LIN {X 0,Y 119.858,Z 319.555,A -85,B 0,C 180,E1 -30049.333,E2 -30049.333} C_VEL
LIN {X 0,Y 123.743,Z 306.108,A -85,B 0,C 180,E1 -30049.858,E2 -30049.858} C_VEL
LIN {X 0,Y 124.732,Z 301.362,A -85,B 0,C 180,E1 -30050.064,E2 -30050.064} C_VEL
LIN {X 0,Y 124.129,Z 298.09,A -85,B 0,C 180,E1 -30054.11,E2 -30054.11} C_VEL
LIN {X 0,Y 123.862,Z 295.451,A -85,B 0,C 180,E1 -30060,E2 -30060} C_VEL
LIN {X 0,Y 124.197,Z 298.699,A -85,B 0,C 180,E1 -30066.907,E2 -30066.907} C_VEL
LIN {X 0,Y 124.718,Z 301.371,A -85,B 0,C 180,E1 -30070.151,E2 -30070.151} C_VEL
LIN {X 0,Y 121.542,Z 314.132,A -85,B 0,C 180,E1 -30070.596,E2 -30070.596} C_VEL
LIN {X 0,Y 117.209,Z 326.252,A -85,B 0,C 180,E1 -30071.353,E2 -30071.353} C_VEL
LIN {X 0,Y 111.468,Z 338.251,A -85,B 0,C 180,E1 -30072.254,E2 -30072.254} C_VEL
LIN {X 0,Y 104.801,Z 349.276,A -85,B 0,C 180,E1 -30073.511,E2 -30073.511} C_VEL
LIN {X 0,Y 98.169,Z 358.213,A -85,B 0,C 180,E1 -30074.89,E2 -30074.89} C_VEL
LIN {X 0,Y 96.602,Z 360.066,A -85,B 0,C 180,E1 -30075.232,E2 -30075.232} C_VEL
LIN {X 0,Y 92.627,Z 364.399,A -85,B 0,C 180,E1 -30075.737,E2 -30075.737} C_VEL
LIN {X 0,Y 85.256,Z 371.05,A -85,B 0,C 180,E1 -30075.683,E2 -30075.683} C_VEL
LIN {X 0,Y 77.46,Z 377.142,A -85,B 0,C 180,E1 -30075.805,E2 -30075.805} C_VEL
LIN {X 0,Y 72.841,Z 380.518,A -85,B 0,C 180,E1 -30076.777,E2 -30076.777} C_VEL
LIN {X 0,Y 63.694,Z 386.573,A -85,B 0,C 180,E1 -30080.311,E2 -30080.311} C_VEL
LIN {X 0,Y 54.383,Z 391.666,A -85,B 0,C 180,E1 -30085.238,E2 -30085.238} C_VEL
LIN {X 0,Y 45.566,Z 395.622,A -85,B 0,C 180,E1 -30091.98,E2 -30091.98} C_VEL
LIN {X 0,Y 37.753,Z 398.542,A -85,B 0,C 180,E1 -30101.882,E2 -30101.882} C_VEL
LIN {X 0,Y 33.345,Z 399.934,A -85,B 0,C 180,E1 -30110.787,E2 -30110.787} C_VEL
LIN {X 0,Y 29.898,Z 400.925,A -85,B 0,C 180,E1 -30121.964,E2 -30121.964} C_VEL
LIN {X 0,Y 27.084,Z 401.756,A -85,B 0,C 180,E1 -30150.006,E2 -30150.006} C_VEL
LIN {X 0,Y 27.692,Z 401.557,A -85,B 0,C 180,E1 -30164.708,E2 -30164.708} C_VEL
LIN {X 0,Y 29.899,Z 400.965,A -85,B 0,C 180,E1 -30178.048,E2 -30178.048} C_VEL
LIN {X 0,Y 37.747,Z 398.621,A -85,B 0,C 180,E1 -30198.143,E2 -30198.143} C_VEL
LIN {X 0,Y 45.549,Z 395.733,A -85,B 0,C 180,E1 -30208.067,E2 -30208.067} C_VEL
LIN {X 0,Y 54.363,Z 391.816,A -85,B 0,C 180,E1 -30214.822,E2 -30214.822} C_VEL
LIN {X 0,Y 63.677,Z 386.766,A -85,B 0,C 180,E1 -30219.745,E2 -30219.745} C_VEL
LIN {X 0,Y 73.296,Z 380.406,A -85,B 0,C 180,E1 -30223.511,E2 -30223.511} C_VEL
LIN {X 0,Y 83.126,Z 372.457,A -85,B 0,C 180,E1 -30226.482,E2 -30226.482} C_VEL
LIN {X 0,Y 93.192,Z 362.567,A -85,B 0,C 180,E1 -30228.636,E2 -30228.636} C_VEL
LIN {X 0,Y 101.655,Z 352.177,A -85,B 0,C 180,E1 -30230.129,E2 -30230.129} C_VEL
LIN {X 0,Y 109.313,Z 340.466,A -85,B 0,C 180,E1 -30231.304,E2 -30231.304} C_VEL
LIN {X 0,Y 115.288,Z 328.776,A -85,B 0,C 180,E1 -30232.11,E2 -30232.11} C_VEL
LIN {X 0,Y 119.884,Z 316.966,A -85,B 0,C 180,E1 -30232.67,E2 -30232.67} C_VEL
LIN {X 0,Y 122.909,Z 306.336,A -85,B 0,C 180,E1 -30233.121,E2 -30233.121} C_VEL
LIN {X 0,Y 122.769,Z 304.591,A -85,B 0,C 180,E1 -30235.896,E2 -30235.896} C_VEL
LIN {X 0,Y 122.833,Z 303.055,A -85,B 0,C 180,E1 -30240,E2 -30240} C_VEL
LIN {X 0,Y 122.855,Z 305.465,A -85,B 0,C 180,E1 -30245.539,E2 -30245.539} C_VEL
LIN {X 0,Y 122.934,Z 306.392,A -85,B 0,C 180,E1 -30246.818,E2 -30246.818} C_VEL
LIN {X 0,Y 119.051,Z 319.603,A -85,B 0,C 180,E1 -30247.302,E2 -30247.302} C_VEL
LIN {X 0,Y 114.106,Z 331.478,A -85,B 0,C 180,E1 -30247.858,E2 -30247.858} C_VEL
LIN {X 0,Y 107.541,Z 343.596,A -85,B 0,C 180,E1 -30248.716,E2 -30248.716} C_VEL
LIN {X 0,Y 99.871,Z 354.762,A -85,B 0,C 180,E1 -30249.87,E2 -30249.87} C_VEL
LIN {X 0,Y 91.405,Z 364.671,A -85,B 0,C 180,E1 -30251.38,E2 -30251.38} C_VEL
LIN {X 0,Y 81.351,Z 374.276,A -85,B 0,C 180,E1 -30253.61,E2 -30253.61} C_VEL
LIN {X 0,Y 71.482,Z 381.916,A -85,B 0,C 180,E1 -30256.539,E2 -30256.539} C_VEL
LIN {X 0,Y 62.526,Z 387.71,A -85,B 0,C 180,E1 -30260.241,E2 -30260.241} C_VEL
LIN {X 0,Y 51.135,Z 393.654,A -85,B 0,C 180,E1 -30266.698,E2 -30266.698} C_VEL
LIN {X 0,Y 42.552,Z 397.231,A -85,B 0,C 180,E1 -30274.324,E2 -30274.324} C_VEL
LIN {X 0,Y 37.428,Z 399.073,A -85,B 0,C 180,E1 -30281.309,E2 -30281.309} C_VEL
LIN {X 0,Y 29.679,Z 401.443,A -85,B 0,C 180,E1 -30301.726,E2 -30301.726} C_VEL
LIN {X 0,Y 27.578,Z 402.044,A -85,B 0,C 180,E1 -30315.23,E2 -30315.23} C_VEL
LIN {X 0,Y 27.017,Z 402.251,A -85,B 0,C 180,E1 -30329.994,E2 -30329.994} C_VEL
LIN {X 0,Y 27.577,Z 402.023,A -85,B 0,C 180,E1 -30344.758,E2 -30344.758} C_VEL
LIN {X 0,Y 29.678,Z 401.408,A -85,B 0,C 180,E1 -30358.262,E2 -30358.262} C_VEL
LIN {X 0,Y 33.057,Z 400.407,A -85,B 0,C 180,E1 -30369.62,E2 -30369.62} C_VEL
LIN {X 0,Y 37.427,Z 399.003,A -85,B 0,C 180,E1 -30378.679,E2 -30378.679} C_VEL
LIN {X 0,Y 45.329,Z 396.066,A -85,B 0,C 180,E1 -30388.501,E2 -30388.501} C_VEL
LIN {X 0,Y 54.111,Z 392.092,A -85,B 0,C 180,E1 -30395.381,E2 -30395.381} C_VEL
LIN {X 0,Y 64.611,Z 386.273,A -85,B 0,C 180,E1 -30400.708,E2 -30400.708} C_VEL
LIN {X 0,Y 74.738,Z 379.307,A -85,B 0,C 180,E1 -30404.536,E2 -30404.536} C_VEL
LIN {X 0,Y 84.675,Z 371.03,A -85,B 0,C 180,E1 -30407.209,E2 -30407.209} C_VEL
LIN {X 0,Y 93.082,Z 362.531,A -85,B 0,C 180,E1 -30408.959,E2 -30408.959} C_VEL
LIN {X 0,Y 101.56,Z 352.031,A -85,B 0,C 180,E1 -30410.418,E2 -30410.418} C_VEL
LIN {X 0,Y 109.251,Z 340.203,A -85,B 0,C 180,E1 -30411.496,E2 -30411.496} C_VEL
LIN {X 0,Y 115.146,Z 328.502,A -85,B 0,C 180,E1 -30412.244,E2 -30412.244} C_VEL
LIN {X 0,Y 119.879,Z 316.102,A -85,B 0,C 180,E1 -30412.807,E2 -30412.807} C_VEL
LIN {X 0,Y 122.665,Z 306.102,A -85,B 0,C 180,E1 -30413.163,E2 -30413.163} C_VEL
LIN {X 0,Y 122.509,Z 304.37,A -85,B 0,C 180,E1 -30415.888,E2 -30415.888} C_VEL
LIN {X 0,Y 122.58,Z 302.578,A -85,B 0,C 180,E1 -30420,E2 -30420} C_VEL
LIN {X 0,Y 122.58,Z 305.293,A -85,B 0,C 180,E1 -30425.965,E2 -30425.965} C_VEL
LIN {X 0,Y 122.633,Z 306.102,A -85,B 0,C 180,E1 -30427.013,E2 -30427.013} C_VEL
LIN {X 0,Y 119.005,Z 318.553,A -85,B 0,C 180,E1 -30427.448,E2 -30427.448} C_VEL
LIN {X 0,Y 114.142,Z 330.578,A -85,B 0,C 180,E1 -30428.163,E2 -30428.163} C_VEL
LIN {X 0,Y 108.476,Z 341.312,A -85,B 0,C 180,E1 -30428.895,E2 -30428.895} C_VEL
LIN {X 0,Y 100.82,Z 352.87,A -85,B 0,C 180,E1 -30430.075,E2 -30430.075} C_VEL
LIN {X 0,Y 93.211,Z 362.184,A -85,B 0,C 180,E1 -30431.441,E2 -30431.441} C_VEL
LIN {X 0,Y 84.828,Z 370.668,A -85,B 0,C 180,E1 -30433.238,E2 -30433.238} C_VEL
LIN {X 0,Y 74.96,Z 378.924,A -85,B 0,C 180,E1 -30436.065,E2 -30436.065} C_VEL
LIN {X 0,Y 72.841,Z 380.518,A -85,B 0,C 180,E1 -30436.777,E2 -30436.777} C_VEL
LIN {X 0,Y 68.081,Z 383.726,A -85,B 0,C 180,E1 -30437.92,E2 -30437.92} C_VEL
LIN {X 0,Y 59.396,Z 388.459,A -85,B 0,C 180,E1 -30438.633,E2 -30438.633} C_VEL
LIN {X 0,Y 50.354,Z 392.477,A -85,B 0,C 180,E1 -30439.651,E2 -30439.651} C_VEL
LIN {X 0,Y 45.103,Z 394.564,A -85,B 0,C 180,E1 -30441.793,E2 -30441.793} C_VEL
LIN {X 0,Y 39.18,Z 396.752,A -85,B 0,C 180,E1 -30446.263,E2 -30446.263} C_VEL
LIN {X 0,Y 33.422,Z 398.607,A -85,B 0,C 180,E1 -30452.752,E2 -30452.752} C_VEL
LIN {X 0,Y 28.201,Z 400,A -85,B 0,C 180,E1 -30461.625,E2 -30461.625} C_VEL
LIN {X 0,Y 23.871,Z 400.99,A -85,B 0,C 180,E1 -30473.936,E2 -30473.936} C_VEL
LIN {X 0,Y 19.993,Z 401.821,A -85,B 0,C 180,E1 -30510.009,E2 -30510.009} C_VEL
LIN {X 0,Y 20.915,Z 401.621,A -85,B 0,C 180,E1 -30529.643,E2 -30529.643} C_VEL
LIN {X 0,Y 23.872,Z 401.029,A -85,B 0,C 180,E1 -30546.08,E2 -30546.08} C_VEL
LIN {X 0,Y 33.417,Z 398.686,A -85,B 0,C 180,E1 -30567.279,E2 -30567.279} C_VEL
LIN {X 0,Y 42.218,Z 395.798,A -85,B 0,C 180,E1 -30576.294,E2 -30576.294} C_VEL
LIN {X 0,Y 51.737,Z 391.88,A -85,B 0,C 180,E1 -30581.974,E2 -30581.974} C_VEL
LIN {X 0,Y 61.581,Z 386.83,A -85,B 0,C 180,E1 -30585.953,E2 -30585.953} C_VEL
LIN {X 0,Y 71.602,Z 380.47,A -85,B 0,C 180,E1 -30588.98,E2 -30588.98} C_VEL
LIN {X 0,Y 81.756,Z 372.52,A -85,B 0,C 180,E1 -30591.338,E2 -30591.338} C_VEL
LIN {X 0,Y 92.055,Z 362.629,A -85,B 0,C 180,E1 -30592.982,E2 -30592.982} C_VEL
LIN {X 0,Y 100.681,Z 352.239,A -85,B 0,C 180,E1 -30594.111,E2 -30594.111} C_VEL
LIN {X 0,Y 108.466,Z 340.526,A -85,B 0,C 180,E1 -30595.019,E2 -30595.019} C_VEL
LIN {X 0,Y 114.706,Z 328.435,A -85,B 0,C 180,E1 -30595.637,E2 -30595.637} C_VEL
LIN {X 0,Y 119.751,Z 315.33,A -85,B 0,C 180,E1 -30596.116,E2 -30596.116} C_VEL
LIN {X 0,Y 120.925,Z 311.412,A -85,B 0,C 180,E1 -30596.328,E2 -30596.328} C_VEL
LIN {X 0,Y 121.08,Z 310.072,A -85,B 0,C 180,E1 -30600,E2 -30600} C_VEL
LIN {X 0,Y 120.94,Z 311.447,A -85,B 0,C 180,E1 -30603.605,E2 -30603.605} C_VEL
LIN {X 0,Y 116.62,Z 324.08,A -85,B 0,C 180,E1 -30604.065,E2 -30604.065} C_VEL
LIN {X 0,Y 111.907,Z 334.363,A -85,B 0,C 180,E1 -30604.448,E2 -30604.448} C_VEL
LIN {X 0,Y 104.96,Z 346.241,A -85,B 0,C 180,E1 -30605.113,E2 -30605.113} C_VEL
LIN {X 0,Y 97.171,Z 356.84,A -85,B 0,C 180,E1 -30606.016,E2 -30606.016} C_VEL
LIN {X 0,Y 88.549,Z 366.391,A -85,B 0,C 180,E1 -30607.2,E2 -30607.2} C_VEL
LIN {X 0,Y 78.271,Z 375.58,A -85,B 0,C 180,E1 -30608.991,E2 -30608.991} C_VEL
LIN {X 0,Y 68.112,Z 382.971,A -85,B 0,C 180,E1 -30611.403,E2 -30611.403} C_VEL
LIN {X 0,Y 58.133,Z 388.905,A -85,B 0,C 180,E1 -30614.719,E2 -30614.719} C_VEL
LIN {X 0,Y 48.353,Z 393.59,A -85,B 0,C 180,E1 -30619.127,E2 -30619.127} C_VEL
LIN {X 0,Y 38.99,Z 397.167,A -85,B 0,C 180,E1 -30625.67,E2 -30625.67} C_VEL
LIN {X 0,Y 33.154,Z 399.009,A -85,B 0,C 180,E1 -30632.007,E2 -30632.007} C_VEL
LIN {X 0,Y 23.66,Z 401.378,A -85,B 0,C 180,E1 -30653.545,E2 -30653.545} C_VEL
LIN {X 0,Y 20.788,Z 401.979,A -85,B 0,C 180,E1 -30670.232,E2 -30670.232} C_VEL
LIN {X 0,Y 19.936,Z 402.186,A -85,B 0,C 180,E1 -30689.991,E2 -30689.991} C_VEL
LIN {X 0,Y 20.787,Z 401.957,A -85,B 0,C 180,E1 -30709.752,E2 -30709.752} C_VEL
LIN {X 0,Y 23.658,Z 401.342,A -85,B 0,C 180,E1 -30726.44,E2 -30726.44} C_VEL
LIN {X 0,Y 27.941,Z 400.341,A -85,B 0,C 180,E1 -30738.978,E2 -30738.978} C_VEL
LIN {X 0,Y 33.152,Z 398.937,A -85,B 0,C 180,E1 -30747.981,E2 -30747.981} C_VEL
LIN {X 0,Y 42.044,Z 395.999,A -85,B 0,C 180,E1 -30756.82,E2 -30756.82} C_VEL
LIN {X 0,Y 51.554,Z 392.026,A -85,B 0,C 180,E1 -30762.588,E2 -30762.588} C_VEL
LIN {X 0,Y 61.869,Z 386.661,A -85,B 0,C 180,E1 -30766.619,E2 -30766.619} C_VEL
LIN {X 0,Y 71.468,Z 380.473,A -85,B 0,C 180,E1 -30769.516,E2 -30769.516} C_VEL
LIN {X 0,Y 81.679,Z 372.449,A -85,B 0,C 180,E1 -30771.669,E2 -30771.669} C_VEL
LIN {X 0,Y 90.263,Z 364.268,A -85,B 0,C 180,E1 -30773.063,E2 -30773.063} C_VEL
LIN {X 0,Y 98.887,Z 354.286,A -85,B 0,C 180,E1 -30774.232,E2 -30774.232} C_VEL
LIN {X 0,Y 106.695,Z 342.991,A -85,B 0,C 180,E1 -30775.023,E2 -30775.023} C_VEL
LIN {X 0,Y 112.768,Z 331.918,A -85,B 0,C 180,E1 -30775.644,E2 -30775.644} C_VEL
LIN {X 0,Y 117.87,Z 319.915,A -85,B 0,C 180,E1 -30776.106,E2 -30776.106} C_VEL
LIN {X 0,Y 120.679,Z 311.152,A -85,B 0,C 180,E1 -30776.382,E2 -30776.382} C_VEL
LIN {X 0,Y 120.856,Z 309.624,A -85,B 0,C 180,E1 -30780,E2 -30780} C_VEL
LIN {X 0,Y 120.636,Z 311.232,A -85,B 0,C 180,E1 -30783.818,E2 -30783.818} C_VEL
LIN {X 0,Y 116.339,Z 323.817,A -85,B 0,C 180,E1 -30784.28,E2 -30784.28} C_VEL
LIN {X 0,Y 111.077,Z 335.229,A -85,B 0,C 180,E1 -30784.815,E2 -30784.815} C_VEL
LIN {X 0,Y 104.142,Z 346.85,A -85,B 0,C 180,E1 -30785.527,E2 -30785.527} C_VEL
LIN {X 0,Y 96.37,Z 357.295,A -85,B 0,C 180,E1 -30786.494,E2 -30786.494} C_VEL
LIN {X 0,Y 88.629,Z 365.833,A -85,B 0,C 180,E1 -30787.628,E2 -30787.628} C_VEL
LIN {X 0,Y 80.081,Z 373.701,A -85,B 0,C 180,E1 -30789.159,E2 -30789.159} C_VEL
LIN {X 0,Y 70.057,Z 381.313,A -85,B 0,C 180,E1 -30791.575,E2 -30791.575} C_VEL
LIN {X 0,Y 61.592,Z 386.64,A -85,B 0,C 180,E1 -30794.112,E2 -30794.112} C_VEL
LIN {X 0,Y 51.757,Z 391.732,A -85,B 0,C 180,E1 -30798.114,E2 -30798.114} C_VEL
LIN {X 0,Y 45.103,Z 394.564,A -85,B 0,C 180,E1 -30801.793,E2 -30801.793} C_VEL
LIN {X 0,Y 39.871,Z 396.435,A -85,B 0,C 180,E1 -30804.577,E2 -30804.577} C_VEL
LIN {X 0,Y 30.579,Z 398.907,A -85,B 0,C 180,E1 -30808.552,E2 -30808.552} C_VEL
LIN {X 0,Y 23.152,Z 400.348,A -85,B 0,C 180,E1 -30813.818,E2 -30813.818} C_VEL
LIN {X 0,Y 18.175,Z 401.13,A -85,B 0,C 180,E1 -30822.554,E2 -30822.554} C_VEL
LIN {X 0,Y 16.811,Z 401.283,A -85,B 0,C 180,E1 -30827.195,E2 -30827.195} C_VEL
LIN {X 0,Y 12.914,Z 401.886,A -85,B 0,C 180,E1 -30870.013,E2 -30870.013} C_VEL
LIN {X 0,Y 14.424,Z 401.686,A -85,B 0,C 180,E1 -30899.173,E2 -30899.173} C_VEL
LIN {X 0,Y 18.598,Z 401.094,A -85,B 0,C 180,E1 -30919.108,E2 -30919.108} C_VEL
LIN {X 0,Y 30.17,Z 398.75,A -85,B 0,C 180,E1 -30938.726,E2 -30938.726} C_VEL
LIN {X 0,Y 39.893,Z 395.862,A -85,B 0,C 180,E1 -30945.694,E2 -30945.694} C_VEL
LIN {X 0,Y 49.995,Z 391.944,A -85,B 0,C 180,E1 -30949.753,E2 -30949.753} C_VEL
LIN {X 0,Y 60.252,Z 386.893,A -85,B 0,C 180,E1 -30952.519,E2 -30952.519} C_VEL
LIN {X 0,Y 70.587,Z 380.533,A -85,B 0,C 180,E1 -30954.663,E2 -30954.663} C_VEL
LIN {X 0,Y 80.991,Z 372.582,A -85,B 0,C 180,E1 -30956.309,E2 -30956.309} C_VEL
LIN {X 0,Y 91.459,Z 362.692,A -85,B 0,C 180,E1 -30957.404,E2 -30957.404} C_VEL
LIN {X 0,Y 100.202,Z 352.3,A -85,B 0,C 180,E1 -30958.148,E2 -30958.148} C_VEL
LIN {X 0,Y 108.081,Z 340.587,A -85,B 0,C 180,E1 -30958.771,E2 -30958.771} C_VEL
LIN {X 0,Y 113.837,Z 329.724,A -85,B 0,C 180,E1 -30959.144,E2 -30959.144} C_VEL
LIN {X 0,Y 118.639,Z 317.882,A -85,B 0,C 180,E1 -30959.442,E2 -30959.442} C_VEL
LIN {X 0,Y 118.928,Z 317.019,A -85,B 0,C 180,E1 -30959.577,E2 -30959.577} C_VEL
LIN {X 0,Y 118.908,Z 317.083,A -85,B 0,C 180,E1 -30960.222,E2 -30960.222} C_VEL
LIN {X 0,Y 118.089,Z 319.488,A -85,B 0,C 180,E1 -30960.447,E2 -30960.447} C_VEL
LIN {X 0,Y 113.146,Z 331.152,A -85,B 0,C 180,E1 -30960.689,E2 -30960.689} C_VEL
LIN {X 0,Y 106.32,Z 343.476,A -85,B 0,C 180,E1 -30961.143,E2 -30961.143} C_VEL
LIN {X 0,Y 98.436,Z 354.639,A -85,B 0,C 180,E1 -30961.702,E2 -30961.702} C_VEL
LIN {X 0,Y 89.69,Z 364.546,A -85,B 0,C 180,E1 -30962.456,E2 -30962.456} C_VEL
LIN {X 0,Y 80.962,Z 372.67,A -85,B 0,C 180,E1 -30963.363,E2 -30963.363} C_VEL
LIN {X 0,Y 70.529,Z 380.643,A -85,B 0,C 180,E1 -30964.799,E2 -30964.799} C_VEL
LIN {X 0,Y 59.698,Z 387.279,A -85,B 0,C 180,E1 -30966.991,E2 -30966.991} C_VEL
LIN {X 0,Y 49.897,Z 392.099,A -85,B 0,C 180,E1 -30969.603,E2 -30969.603} C_VEL
LIN {X 0,Y 39.789,Z 396.036,A -85,B 0,C 180,E1 -30973.708,E2 -30973.708} C_VEL
LIN {X 0,Y 29.991,Z 398.944,A -85,B 0,C 180,E1 -30980.374,E2 -30980.374} C_VEL
LIN {X 0,Y 18.419,Z 401.313,A -85,B 0,C 180,E1 -31000.246,E2 -31000.246} C_VEL
LIN {X 0,Y 14.295,Z 401.914,A -85,B 0,C 180,E1 -31020.538,E2 -31020.538} C_VEL
LIN {X 0,Y 12.841,Z 402.121,A -85,B 0,C 180,E1 -31049.986,E2 -31049.986} C_VEL
LIN {X 0,Y 14.292,Z 401.892,A -85,B 0,C 180,E1 -31079.44,E2 -31079.44} C_VEL
LIN {X 0,Y 18.416,Z 401.277,A -85,B 0,C 180,E1 -31099.737,E2 -31099.737} C_VEL
LIN {X 0,Y 23.881,Z 400.275,A -85,B 0,C 180,E1 -31111.973,E2 -31111.973} C_VEL
LIN {X 0,Y 29.986,Z 398.871,A -85,B 0,C 180,E1 -31119.615,E2 -31119.615} C_VEL
LIN {X 0,Y 39.783,Z 395.933,A -85,B 0,C 180,E1 -31126.294,E2 -31126.294} C_VEL
LIN {X 0,Y 49.89,Z 391.96,A -85,B 0,C 180,E1 -31130.403,E2 -31130.403} C_VEL
LIN {X 0,Y 61.488,Z 386.08,A -85,B 0,C 180,E1 -31133.437,E2 -31133.437} C_VEL
LIN {X 0,Y 72.255,Z 379.173,A -85,B 0,C 180,E1 -31135.496,E2 -31135.496} C_VEL
LIN {X 0,Y 82.698,Z 370.895,A -85,B 0,C 180,E1 -31136.867,E2 -31136.867} C_VEL
LIN {X 0,Y 91.43,Z 362.395,A -85,B 0,C 180,E1 -31137.744,E2 -31137.744} C_VEL
LIN {X 0,Y 100.18,Z 351.893,A -85,B 0,C 180,E1 -31138.463,E2 -31138.463} C_VEL
LIN {X 0,Y 108.068,Z 340.063,A -85,B 0,C 180,E1 -31138.958,E2 -31138.958} C_VEL
LIN {X 0,Y 114.469,Z 327.524,A -85,B 0,C 180,E1 -31139.342,E2 -31139.342} C_VEL
LIN {X 0,Y 118.391,Z 317.575,A -85,B 0,C 180,E1 -31139.587,E2 -31139.587} C_VEL
LIN {X 0,Y 118.725,Z 316.57,A -85,B 0,C 180,E1 -31140,E2 -31140} C_VEL
LIN {X 0,Y 118.692,Z 316.668,A -85,B 0,C 180,E1 -31140.424,E2 -31140.424} C_VEL
LIN {X 0,Y 116.544,Z 322.553,A -85,B 0,C 180,E1 -31140.733,E2 -31140.733} C_VEL
LIN {X 0,Y 111.585,Z 333.578,A -85,B 0,C 180,E1 -31141.111,E2 -31141.111} C_VEL
LIN {X 0,Y 105.45,Z 344.299,A -85,B 0,C 180,E1 -31141.497,E2 -31141.497} C_VEL
LIN {X 0,Y 97.575,Z 355.227,A -85,B 0,C 180,E1 -31142.127,E2 -31142.127} C_VEL
LIN {X 0,Y 89.712,Z 364.121,A -85,B 0,C 180,E1 -31142.842,E2 -31142.842} C_VEL
LIN {X 0,Y 80.998,Z 372.286,A -85,B 0,C 180,E1 -31143.834,E2 -31143.834} C_VEL
LIN {X 0,Y 70.595,Z 380.287,A -85,B 0,C 180,E1 -31145.454,E2 -31145.454} C_VEL
LIN {X 0,Y 60.257,Z 386.706,A -85,B 0,C 180,E1 -31147.561,E2 -31147.561} C_VEL
LIN {X 0,Y 50.004,Z 391.799,A -85,B 0,C 180,E1 -31150.341,E2 -31150.341} C_VEL
LIN {X 0,Y 39.898,Z 395.754,A -85,B 0,C 180,E1 -31154.371,E2 -31154.371} C_VEL
LIN {X 0,Y 30.171,Z 398.673,A -85,B 0,C 180,E1 -31161.311,E2 -31161.311} C_VEL
LIN {X 0,Y 24.07,Z 400.065,A -85,B 0,C 180,E1 -31168.86,E2 -31168.86} C_VEL
LIN {X 0,Y 16.811,Z 401.283,A -85,B 0,C 180,E1 -31187.195,E2 -31187.195} C_VEL
LIN {X 0,Y 14.326,Z 401.634,A -85,B 0,C 180,E1 -31198.427,E2 -31198.427} C_VEL
LIN {X 0,Y 11.106,Z 401.882,A -85,B 0,C 180,E1 -31221.167,E2 -31221.167} C_VEL
LIN {X 0,Y 13.108,Z 401.433,A -85,B 0,C 180,E1 -31291.269,E2 -31291.269} C_VEL
LIN {X 0,Y 18.867,Z 400.633,A -85,B 0,C 180,E1 -31305.47,E2 -31305.47} C_VEL
LIN {X 0,Y 19.8,Z 400.438,A -85,B 0,C 180,E1 -31306.472,E2 -31306.472} C_VEL
LIN {X 0,Y 28.371,Z 398.815,A -85,B 0,C 180,E1 -31312.284,E2 -31312.284} C_VEL
LIN {X 0,Y 38.754,Z 395.926,A -85,B 0,C 180,E1 -31315.937,E2 -31315.937} C_VEL
LIN {X 0,Y 49.229,Z 392.008,A -85,B 0,C 180,E1 -31317.951,E2 -31317.951} C_VEL
LIN {X 0,Y 58.335,Z 387.683,A -85,B 0,C 180,E1 -31319.141,E2 -31319.141} C_VEL
LIN {X 0,Y 60.788,Z 386.385,A -85,B 0,C 180,E1 -31320,E2 -31320} C_VEL
LIN {X 0,Y 49.213,Z 392.035,A -85,B 0,C 180,E1 -31321.417,E2 -31321.417} C_VEL
LIN {X 0,Y 38.725,Z 395.972,A -85,B 0,C 180,E1 -31323.419,E2 -31323.419} C_VEL
LIN {X 0,Y 28.309,Z 398.879,A -85,B 0,C 180,E1 -31326.718,E2 -31326.718} C_VEL
LIN {X 0,Y 14.849,Z 401.249,A -85,B 0,C 180,E1 -31338.78,E2 -31338.78} C_VEL
LIN {X 0,Y 8.828,Z 401.85,A -85,B 0,C 180,E1 -31357.214,E2 -31357.214} C_VEL
LIN {X 0,Y 5.738,Z 402.056,A -85,B 0,C 180,E1 -31409.97,E2 -31409.97} C_VEL
LIN {X 0,Y 8.824,Z 401.827,A -85,B 0,C 180,E1 -31462.759,E2 -31462.759} C_VEL
LIN {X 0,Y 14.844,Z 401.212,A -85,B 0,C 180,E1 -31481.205,E2 -31481.205} C_VEL
LIN {X 0,Y 21.473,Z 400.21,A -85,B 0,C 180,E1 -31489.021,E2 -31489.021} C_VEL
LIN {X 0,Y 28.303,Z 398.805,A -85,B 0,C 180,E1 -31493.273,E2 -31493.273} C_VEL
LIN {X 0,Y 38.719,Z 395.867,A -85,B 0,C 180,E1 -31496.584,E2 -31496.584} C_VEL
LIN {X 0,Y 49.207,Z 391.893,A -85,B 0,C 180,E1 -31498.588,E2 -31498.588} C_VEL
LIN {X 0,Y 60.699,Z 386.235,A -85,B 0,C 180,E1 -31500.054,E2 -31500.054} C_VEL
LIN {X 0,Y 63.249,Z 384.77,A -85,B 0,C 180,E1 -31500.44,E2 -31500.44} C_VEL
LIN {X 0,Y 52.726,Z 390.277,A -85,B 0,C 180,E1 -31501.598,E2 -31501.598} C_VEL
LIN {X 0,Y 42.237,Z 394.597,A -85,B 0,C 180,E1 -31503.364,E2 -31503.364} C_VEL
LIN {X 0,Y 35.272,Z 396.884,A -85,B 0,C 180,E1 -31505.03,E2 -31505.03} C_VEL
LIN {X 0,Y 28.368,Z 398.739,A -85,B 0,C 180,E1 -31507.76,E2 -31507.76} C_VEL
LIN {X 0,Y 21.553,Z 400.131,A -85,B 0,C 180,E1 -31512.026,E2 -31512.026} C_VEL
LIN {X 0,Y 12.19,Z 401.385,A -85,B 0,C 180,E1 -31525.545,E2 -31525.545} C_VEL
LIN {X 0,Y 5.821,Z 401.95,A -85,B 0,C 180,E1 -31590.03,E2 -31590.03} C_VEL
LIN {X 0,Y 8.926,Z 401.751,A -85,B 0,C 180,E1 -31641.968,E2 -31641.968} C_VEL
LIN {X 0,Y 19.8,Z 400.438,A -85,B 0,C 180,E1 -31666.472,E2 -31666.472} C_VEL
LIN {X 0,Y 21.97,Z 402.419,A -85,B 0,C 180,E1 -31668.335,E2 -31668.335} C_VEL
LIN {X 0,Y 21.97,Z 600,A -85,B 0,C 180,E1 -31668.335,E2 -31668.335} C_VEL
LIN {X 0,Y 21.97,Z 600,A -85,B 0,C 180,E1 -31668.335,E2 -31668.335}

QRS_NEXT_CUT()

QRS_NEXT()
QRS_HOME()

END
